{attribute 'GeneratedUsingTerminal: KL6211-0004'}
{attribute addProperty BoxType "KL6211-0004"}
{attribute addProperty Description ""}
{attribute addProperty Physics ""}
{attribute addProperty Id "Channel_1AT %Q*Channel_A6A8AB450"}
{attribute addProperty CRC "1899239057"}
{attribute addProperty Size "0"}
TYPE KL_71341691 :
STRUCT
	{attribute addProperty Name "Channel_1"}
	Channel_1 : Channel_A6A8AB45;
END_STRUCT
END_TYPE

(* stored: Version 1.2.0.0, ProductVersion 3.1.4024.9
   DUT KL_71341691: Id {173715f0-569e-42d7-8f98-777829aca016} *)
